// TwinCAT 3 PLC project PLC1
// ProgramVersion: 3.1.4024.0
// libraries:
//   Tc2_Standard, * (Beckhoff Automation GmbH)
//   Tc2_System, * (Beckhoff Automation GmbH)
//   Tc3_Module, * (Beckhoff Automation GmbH)
// project tree:
//   GVLs/ GVL_Safety.TcGVL
//   / PlcTask.TcTTO
//   POUs/ FB_Clock.TcPOU (not stored), MAIN.TcPOU
// real-time tasks:
//   TASK PlcTask: cycle T#10ms, priority 20, ADS port 350
// I/O:
//   DEVICE Device 3 (EtherCAT), AmsNetId 192.168.137.33.4.1
//     Term 1 (EK1100) [EK1100 EtherCAT Coupler (2A E-Bus)]
//       Term 2 (EK1122) [EK1122 2 port EtherCAT junction]
//         Term 3 (EK1960-0000) [EK1960-0000 TwinSAFE-Compact-Controller (RJ45)]
//           modules: Module 2 (FSOUT), Module 3 (FSLOGIC)
//         Term 4 (EK1960-2600) [EK1960-2600 TwinSAFE-Compact-Controller (4 x Relay, RJ45)]
//           modules: Module 2 (FSOUT), Module 3 (FSLOGIC)
// variable links:
//   Device 3 (EtherCAT) <-> Device 3 (EtherCAT)/Term 1 (EK1100)/Term 2 (EK1122)/Term 4 (EK1960-2600)
//     Term 1 (EK1100)/Term 2 (EK1122)/Term 3 (EK1960-0000)/ConnectionInputs/Message_9 TxPDO <-> ConnectionOutputs/Message_6 RxPDO
//     Term 1 (EK1100)/Term 2 (EK1122)/Term 3 (EK1960-0000)/ConnectionOutputs/Message_9 RxPDO <-> ConnectionInputs/Message_6 TxPDO
//   PLC1/PLC1 Instance <-> Device 3 (EtherCAT)
//     PlcTask Inputs/MAIN.infoData <-> Inputs/SlaveCount
//   PLC1/PLC1 Instance <-> Device 3 (EtherCAT)/Term 1 (EK1100)/Term 2 (EK1122)/Term 3 (EK1960-0000)
//     PlcTask Outputs/GVL_Safety.bEnableClockEK1960_0000 <-> StandardOutputs/Standard In Var 4
//     PlcTask Outputs/GVL_Safety.bRunEK1960_0000 <-> StandardOutputs/Standard In Var 10
//   PLC1/PLC1 Instance <-> Device 3 (EtherCAT)/Term 1 (EK1100)/Term 2 (EK1122)/Term 4 (EK1960-2600)
//     PlcTask Outputs/GVL_Safety.bEnableClockEK1960_2600 <-> StandardOutputs/Standard In Var 8
//     PlcTask Outputs/GVL_Safety.bRunEK1960_2600 <-> StandardOutputs/Standard In Var 7

CONFIGURATION PLC1
    RESOURCE PLC ON TwinCAT3
        TASK PlcTask(INTERVAL := T#10ms, PRIORITY := 20);
        PROGRAM MAIN WITH PlcTask : MAIN;
    END_RESOURCE
END_CONFIGURATION

// ---- GVLs/GVL_Safety.TcGVL
{attribute 'qualified_only'}
VAR_GLOBAL
	bEnableClockEK1960_0000 AT%Q* : BOOL;
	bEnableClockEK1960_2600 AT%Q* : BOOL;
	bRunEK1960_0000 AT%Q* : BOOL;
	bRunEK1960_2600 AT%Q* : BOOL;
END_VAR

// ---- POUs/MAIN.TcPOU
PROGRAM MAIN
VAR
	infoData AT%I* : UINT;
	fbClock1: FB_Clock;
	fbClock2: FB_Clock;
END_VAR

fbClock1(TIME_ON:= T#1S, TIME_OFF:= T#1S, OUT_CLK=>);
fbClock2(TIME_ON:= T#300MS, TIME_OFF:= T#300MS, OUT_CLK=>);
GVL_safety.bEnableClockEK1960_0000 := fbClock1.OUT_CLK;
GVL_safety.bEnableClockEK1960_2600 := fbClock2.OUT_CLK;

END_PROGRAM
